// TwinCAT 3 PLC project Tc_Math
// Title: Tc_Math
// Company: NewEngineer
// Author: https://github.com/phucpha
// ProjectVersion: 1.1.2.0
// Description: this is library expand the Tc2_math
// ProgramVersion: 3.1.4024.0
// libraries:
//   Tc2_Math, * (Beckhoff Automation GmbH)
//   Tc2_Standard, * (Beckhoff Automation GmbH)
//   Tc2_System, * (Beckhoff Automation GmbH)
//   Tc2_Utilities, * (Beckhoff Automation GmbH)
//   Tc3_Module, * (Beckhoff Automation GmbH)
// project tree:
//   DUTs/ E_CompareTime.TcDUT
//   FCs/ F_CompareTime.TcPOU, FUN_Ceil.TcPOU, F_CheckInRange.TcPOU (not stored), F_CubicFit.TcPOU, F_CubitCalculate.TcPOU (not stored), F_InRange.TcPOU (not stored), F_QuanDraticCalculate.TcPOU (not stored), F_QuandraticFomularMaxValue.TcPOU, F_RoundLrealEx.TcPOU, F_ScaleValue.TcPOU (not stored)
//   / PlcTask.TcTTO
//   POUs/ FB_CalCulateAccumulation.TcPOU, FB_Derivative.TcPOU (not stored)
//   POUs/FIFO/ FB_FIFO_Lreal.TcPOU, FB_FIFO_TimeStruct.TcPOU, FB_Universal_FIFO.TcPOU, I_FIFO_Lreal.TcIO, I_FIFO_Timestruct.TcIO, I_Universal_FIFO.TcIO
// real-time tasks:
//   TASK PlcTask: cycle T#10ms, priority 20, ADS port 350

CONFIGURATION Tc_Math
    RESOURCE PLC ON TwinCAT3
        TASK PlcTask(INTERVAL := T#10ms, PRIORITY := 20);
    END_RESOURCE
END_CONFIGURATION

// ---- DUTs/E_CompareTime.TcDUT
{attribute 'strict'}
TYPE E_CompareTime :
(
	INVALID_PRE_TIME := 0,
	NEW_MINUTE := 5,
	NEW_HOUR := 10,
	NEW_DAY	:= 20,
	NEW_MONTH := 30,
	NEW_YEAR	:= 32,
	SAME_MINUTE := 35,
	SAME_HOUR := 40,
	SAME_DAY := 50,
	SAME_MONTH := 60,
	SAME_YEAR  := 70
);
END_TYPE

// ---- POUs/FIFO/I_FIFO_Lreal.TcIO
INTERFACE I_FIFO_Lreal EXTENDS I_Universal_FIFO

METHOD MR_AddValue : BOOL
VAR_INPUT
		Value : LREAL;
END_VAR
END_METHOD

PROPERTY oOldestValue : Lreal
GET
END_GET
END_PROPERTY

END_INTERFACE

// ---- POUs/FIFO/I_FIFO_Timestruct.TcIO
INTERFACE I_FIFO_Timestruct EXTENDS I_Universal_FIFO

METHOD MR_AddValue : BOOL
VAR_INPUT
		Value : TIMESTRUCT;
END_VAR
END_METHOD

PROPERTY oOldestValue : TIMESTRUCT
GET
END_GET
END_PROPERTY

END_INTERFACE

// ---- POUs/FIFO/I_Universal_FIFO.TcIO
INTERFACE I_Universal_FIFO

PROPERTY DataReady : bool
GET
END_GET
END_PROPERTY

PROPERTY HeadIndex : Uint
GET
END_GET
END_PROPERTY

PROPERTY IsEmpty : bool
GET
END_GET
END_PROPERTY

PROPERTY IsFull : bool
GET
END_GET
END_PROPERTY

METHOD MR_AckGetValue : BOOL
VAR_INPUT
END_VAR
END_METHOD

METHOD MR_Reset : BOOL
VAR_INPUT
END_VAR
END_METHOD

PROPERTY TailIndex : Uint
GET
END_GET
END_PROPERTY

END_INTERFACE

// ---- FCs/F_CompareTime.TcPOU
FUNCTION F_CompareTime : E_CompareTime
VAR_INPUT
		timestruct1 : TIMESTRUCT;//TIMEPREVIOUS
		timestruct2 : TIMESTRUCT;// TIME NOW
END_VAR
VAR_OUTPUT
	eCpMinute	: E_CompareTime;
	eCpHour		: E_CompareTime;
	eCpDay		: E_CompareTime;
	eCpMonth	: E_CompareTime;
	ecpYear		: E_CompareTime;
END_VAR

IF timestruct1.wYear < timestruct2.wYear THEN
	F_CompareTime := NEW_YEAR;
	ecpYear := NEW_YEAR;
	eCpMonth := NEW_MONTH;
	eCpDay := NEW_DAY;
	eCpHour := NEW_HOUR;
	eCpMinute := NEW_MINUTE;
ELSIF timestruct1.wYear > timestruct2.wYear THEN
		F_CompareTime := INVALID_PRE_TIME;
ELSE 
	ecpYear := SAME_YEAR;
	IF timestruct1.wMonth < timestruct2.wMonth THEN
		F_CompareTime := NEW_MONTH;
		eCpMonth := NEW_MONTH;
		eCpDay := NEW_DAY;
		eCpHour := NEW_HOUR;
		eCpMinute := NEW_MINUTE;
	ELSIF  timestruct1.wMonth > timestruct2.wMonth THEN
			F_CompareTime := INVALID_PRE_TIME;
	ELSE
		eCpMonth := SAME_MONTH;
		IF timestruct1.wDay < timestruct2.wDay THEN
			F_CompareTime := NEW_DAY;
			eCpDay := NEW_DAY;
			eCpHour := NEW_HOUR;
			eCpMinute := NEW_MINUTE;
		ELSIF timestruct1.wDay > timestruct2.wDay THEN
			F_CompareTime := INVALID_PRE_TIME;
		ELSE 
			eCpDay := SAME_DAY;
			IF timestruct1.wHour < timestruct2.wHour THEN
				F_CompareTime := NEW_HOUR;
				eCpHour := NEW_HOUR;
				eCpMinute := NEW_MINUTE;
			ELSIF timestruct1.wHour > timestruct2.wHour THEN
				F_CompareTime := INVALID_PRE_TIME; 
			ELSE
				eCpHour := SAME_HOUR;
				IF timestruct1.wMinute < timestruct2.wMinute THEN
					F_CompareTime := NEW_MINUTE;
					eCpMinute := NEW_MINUTE;
				ELSIF timestruct1.wMinute > timestruct2.wMinute THEN
					F_CompareTime := INVALID_PRE_TIME; 
				ELSE
					F_CompareTime := SAME_MINUTE;	
					eCpMinute := SAME_MINUTE;
			END_IF
			END_IF
		END_IF

	END_IF
END_IF

END_FUNCTION

// ---- FCs/FUN_Ceil.TcPOU
(* 
:Description: This function determines a integral value from a floating point number that is a fraction bigger than or equal that number
*)
FUNCTION FUN_Ceil : LREAL
VAR_INPUT
	lrValue : LREAL; (* Input value to round*)
END_VAR
VAR
	lrIntegral	: LREAL; (* Integral part of input value *)
	lrDecimal 	: LREAL; (* Decimal part of input value *)
END_VAR

(* Get integral part *)
lrIntegral := TRUNC(lrValue);

(* Get decimal part *)
lrDecimal := FRAC(lrValue);

(*Check decimal value and set final result *)
IF lrDecimal <> 0.0 THEN
	FUN_Ceil := lrIntegral + 1.0;
ELSE
	FUN_Ceil := lrIntegral;
END_IF

END_FUNCTION

// ---- FCs/F_CubicFit.TcPOU
FUNCTION F_CubicFit : BOOL
VAR_INPUT
    x : ARRAY[0..3] OF REAL; // x0, x1, x2, x3
    y : ARRAY[0..3] OF REAL; // y0, y1, y2, y3
END_VAR

VAR_OUTPUT
    a, b, c, d : REAL; // Polynomial coefficients
END_VAR

VAR
    Arr : ARRAY[0..3] OF ARRAY [0..4] OF REAL; // Augmented matrix (4x5)
    i, j, k : INT;
    factor : REAL;
END_VAR

// Build the augmented matrix A
FOR i := 0 TO 3 DO
    Arr[i][0] := x[i] * x[i] * x[i]; // x^3
    Arr[i][1] := x[i] * x[i];        // x^2
    Arr[i][2] := x[i];               // x
    Arr[i][3] := 1.0;                // constArrnt
    Arr[i][4] := y[i];               // y value (RHS)
END_FOR

// Gauss-Jordan Elimination
FOR i := 0 TO 3 DO
    // Normalize row i
    factor := Arr[i][ i];
    FOR j := i TO 4 DO
		IF NOT (-0.00000001 < factor  AND factor <  0.00000001) THEN
        	Arr[i][j] := Arr[i][ j] / factor;
		END_IF
    END_FOR

    // Eliminate other rows
    FOR k := 0 TO 3 DO
        IF k <> i THEN
            factor := Arr[k][ i];
            FOR j := i TO 4 DO
                Arr[k][j] := Arr[k][ j] - factor * Arr[i][j];
            END_FOR
        END_IF
    END_FOR
END_FOR

// Extract coefficients
a := Arr[0][ 4];
b := Arr[1][ 4];
c := Arr[2][ 4];
d := Arr[3][ 4];

END_FUNCTION

// ---- FCs/F_QuandraticFomularMaxValue.TcPOU
FUNCTION F_QuandraticFomularMaxValue : LREAL 
VAR_INPUT
	A : LREAL;
	B : LREAL;
	C : LREAL;
	xLimit1 : LREAL;
	xLimit2 : LREAL;
END_VAR
VAR
	yAtxLimit1 : LREAL;
	yAtxLimit2 : LREAL;
	Adot : LREAL; // Adot = A'
	Bdot : LREAL; // Bdot = B'
	x : LREAL;
END_VAR
VAR_OUTPUT
	MaxValue : LREAL;
END_VAR

yAtxLimit1 := F_QuanDraticCalculate(
	A := A,
	B := B,
	C := C,
	x := xLimit1
);
yAtxLimit2 := F_QuanDraticCalculate(
	A := A,
	B := B,
	C := C,
	x := xLimit2
);		
IF A > 0 THEN
	MaxValue := MAX(yAtxLimit1, yAtxLimit2);
ELSIF A < 0 THEN
	Adot := 2 * A;
	Bdot := B;
	x := -Bdot / Adot;
	MaxValue := F_QuanDraticCalculate(
		A := A,
		B := B,
		C := C,
		x := x
	);	
ELSE // A = 0, b is any
	MaxValue := MAX(yAtxLimit1, yAtxLimit2);
END_IF
F_QuandraticFomularMaxValue := MaxValue;

END_FUNCTION

// ---- FCs/F_RoundLrealEx.TcPOU
FUNCTION F_RoundLrealEx : LREAL
VAR_INPUT
	lrIn : LREAL;
	iPrecision : UINT;
END_VAR
VAR
	lrTemp	: LREAL;
END_VAR

lrTemp := lrIn * EXPT(10,iPrecision);
lrTemp := LTRUNC(lrTemp);
F_RoundLrealEx := lrTemp / EXPT(10,iPrecision);

END_FUNCTION

// ---- POUs/FB_CalCulateAccumulation.TcPOU
(* Will be refactor later
| need refactor to independence to fbMachineTime 
*)
FUNCTION_BLOCK FB_CalCulateAccumulation
VAR_INPUT
	lrAccumulator : LREAL  := 0;
	CurrentTime : TIMESTRUCT; 
END_VAR
VAR_OUTPUT
	accumulatedValueOut : LREAL;// value = lrAccumulator(timeNew) - lrAccumulator(timeOld)
	previousTimestampOut : TIMESTRUCT;// TimeOld
	bNewPeriodAlarm : BOOL;// Remain True in 30s if not be ackNowledge
	
END_VAR
VAR

	
	eCpHour		: E_CompareTime;
	eCpDay 		: E_CompareTime;
	eCpMonth	: E_CompareTime;
	eCpYear		: E_CompareTime;
	eCpMinute	: E_CompareTime;
	eSameTime : E_CompareTime;
	eNewTime : E_CompareTime;
	eRfTimeCompare : REFERENCE TO E_CompareTime;
	sName 		: STRING;
	eState : UINT;
	TonRemainOutput : TON;
	eTimeAccumulate : E_CompareTime;
	bInit : BOOL;
	bReset : BOOL;
	bRequestUpdate_ValueInLastTime: BOOL;
END_VAR

VAR PERSISTENT 
	bUpdatedValueLastHour : BOOL;// reject Power OFF unexpected
	previousTimestamp	: TIMESTRUCT;
	ValueInLastTime : LREAL;
	accumulatedValue : LREAL;
	
	
END_VAR
VAR CONSTANT
	eStateUinitialized : UINT := 0;
	eStateInit : UINT := 10;
	eStateRun : UINT := 20;
	eStateReset : UINT := 100;
	TimeNewPeriodAlarm : TIME := T#30s;
END_VAR

CASE eState OF
	eStateUinitialized: // unInitialized
		;// will go to eStateInit if MR_Run is called 
		
	eStateInit: 
		;// will call by MR_Init
		
	eStateRun: //StateRun
		MS_Run();
		
	eStateReset :
		MS_Reset();
END_CASE

IF eState > 0 AND bReset THEN
	eState := eStateReset;
END_IF

PROPERTY isInitDone : bool
GET
END_GET
END_PROPERTY

PROPERTY isRuning : bool
GET
isRuning := eState = eStateRun;
END_GET
END_PROPERTY

// if not return true , check the Current time and PreviousTime in fb
METHOD MR_Acknowledge : BOOL
VAR_INPUT
END_VAR
bNewPeriodAlarm := FALSE;
IF eRfTimeCompare = eSameTime THEN
	MR_Acknowledge := TRUE;
END_IF
END_METHOD

METHOD MR_Init : BOOL
VAR_INPUT
END_VAR
IF eState = eStateUinitialized THEN// init;
	bInit := true;
	IF MS_Init() THEN
		MR_Init := TRUE;
		eState := eStateRun;
	END_IF
END_IF
END_METHOD

METHOD MR_Reset : BOOL
VAR_INPUT
END_VAR
bReset := TRUE;
IF eState = eStateUinitialized THEN
	MR_Reset := TRUE;
	bReset := false;
END_IF
END_METHOD

METHOD Protected MS_Init : BOOL
VAR_INPUT
END_VAR
CASE eTimeAccumulate OF
	NEW_MINUTE :
		eSameTime := SAME_MINUTE;
		eNewTime := NEW_MINUTE;
		eRfTimeCompare REF= eCpMinute;
		MS_Init := TRUE;
	NEW_HOUR :
		eSameTime := SAME_HOUR;
		eNewTime := NEW_HOUR;
		eRfTimeCompare REF= eCpHour;
		MS_Init := TRUE;
	NEW_DAY	:
		eSameTime := SAME_DAY;
		eNewTime := NEW_DAY;
		eRfTimeCompare REF= eCpDay;
		MS_Init := TRUE;
	NEW_MONTH:
		eSameTime := SAME_MONTH;
		eNewTime := NEW_MONTH;
		eRfTimeCompare REF= eCpMonth;
		MS_Init := TRUE;
	NEW_YEAR:
		eSameTime := SAME_YEAR;
		eNewTime := NEW_YEAR;
		eRfTimeCompare REF= eCpYear;
		MS_Init := true;
END_CASE
END_METHOD

METHOD protected MS_Reset : BOOL
VAR_INPUT
END_VAR
//retainvalue
	
	bUpdatedValueLastHour := FALSE;
	previousTimestamp.wYear := 0;
	previousTimestamp.wMonth := 0;
	previousTimestamp.wDay := 0;
	previousTimestamp.wMinute := 0;
	previousTimestamp.wSecond := 0;
	previousTimestamp.wMilliseconds := 0;
	ValueInLastTime := 0 ;
	accumulatedValue := 0 ;
// out_put
	accumulatedValueOut := 0;
	previousTimestampOut.wYear := 0;
	previousTimestampOut.wMonth := 0;
	previousTimestampOut.wDay := 0;
	previousTimestampOut.wMinute := 0;
	previousTimestampOut.wSecond := 0;
	previousTimestampOut.wMilliseconds := 0;
	bNewPeriodAlarm := false;// Remain True 
	
// 	RETURN TO uninit
	eState := eStateUinitialized;
	eRfTimeCompare REF= 0;
END_METHOD

METHOD Protected MS_Run : BOOL
VAR_INPUT
END_VAR
F_CompareTime( 
	timestruct1 := previousTimestamp,
	timestruct2 := CurrentTime,
	eCpMinute => eCpMinute, 
	eCpHour => eCpHour,
	eCpDay => eCpDay,
	eCpMonth => eCpMonth,
	ecpYear => eCpYear
);

IF eRfTimeCompare = eNewTime THEN
	// update to output
	accumulatedValueOut := accumulatedValue;
	previousTimestampOut := previousTimestamp;
	bNewPeriodAlarm := TRUE;
	// update the the last hour and time
	bUpdatedValueLastHour := FALSE;
	IF lrAccumulator > 0.1 THEN
		ValueInLastTime := lrAccumulator;
		bRequestUpdate_ValueInLastTime := FALSE;
		// UpdateOK
		bUpdatedValueLastHour := TRUE;
	ELSE
		bRequestUpdate_ValueInLastTime := TRUE;
	END_IF
	ValueInLastTime := lrAccumulator;
	previousTimestamp := CurrentTime;


ELSIF eRfTimeCompare = eSameTime AND bUpdatedValueLastHour THEN
	IF lrAccumulator > 0.1 THEN // reject the situation that just TURN ON IPC so lrAccumulator = -8888888888888888.444444444444
		accumulatedValue := lrAccumulator - ValueInLastTime;
	END_IF
ELSIF eRfTimeCompare = eSameTime AND NOT bUpdatedValueLastHour THEN
	ValueInLastTime := lrAccumulator;
	previousTimestamp := CurrentTime;
ELSE
	; //invalid time Compare


END_IF
	
TonRemainOutput( IN := bNewPeriodAlarm , PT := TimeNewPeriodAlarm);

IF TonRemainOutput.Q THEN
	bNewPeriodAlarm := false;
END_IF
IF bRequestUpdate_ValueInLastTime THEN
	IF lrAccumulator > 0.1 THEN
		ValueInLastTime := lrAccumulator;
		bRequestUpdate_ValueInLastTime := FALSE;
		// UpdateOK
		bUpdatedValueLastHour := TRUE;
	END_IF
END_IF
END_METHOD

PROPERTY Name : string
GET
Name := sName;
END_GET
SET
sName := Name;
END_SET
END_PROPERTY

// Set TimeAccumulate before call Mr_Init.
//NEW_MINUTE := 5,
//	NEW_HOUR := 10,
//	NEW_DAY	:= 20,
//	NEW_MONTH := 30,
//	NEW_YEAR	:= 32,
PROPERTY TimeAccumulate : E_CompareTime
GET
TimeAccumulate := eTimeAccumulate;
END_GET
SET
eTimeAccumulate := TimeAccumulate;
END_SET
END_PROPERTY

END_FUNCTION_BLOCK

// ---- POUs/FIFO/FB_FIFO_Lreal.TcPOU
FUNCTION_BLOCK FB_FIFO_Lreal EXTENDS FB_Universal_FIFO IMPLEMENTS I_FIFO_Lreal
VAR_OUTPUT
	OldestData : LREAL;
END_VAR
VAR PERSISTENT
	Queue : ARRAY[0..MaxQueueSize-1] OF LREAL;  // FIFO queue (size is 100 elements)
END_VAR



//    // Log new data only if LogData is TRUE
//    IF rTrigLogData.Q THEN
//        IF Count < MaxQueueSize THEN
//            Queue[Head] := NewEnergyData;
//            Head := (Head + 1) MOD MaxQueueSize;
//            Count := Count + 1;
//        ELSE
//            // FIFO is full, overwrite old data if needed
//            Tail := (Tail + 1) MOD MaxQueueSize;
//            Queue[Head] := NewEnergyData;
//            Head := (Head + 1) MOD MaxQueueSize;
//            // Tail position is updated
//        END_IF
//        DataReady := TRUE;  // New data is now ready to be processed
     
//    END_IF

    // Retrieve and manage oldest data for processing

// if dataready return true, else return false
METHOD  MR_AckGetValue : BOOL
VAR_INPUT
END_VAR
SUPER^.MR_AckGetValue();
  OldestData := Queue[Tail];
 MR_AckGetValue := true;
END_METHOD

METHOD MR_AddValue : BOOL
VAR_INPUT
		Value : LREAL;
END_VAR
  IF Count < MaxQueueSize THEN
            Queue[Head] := Value;
            Head := (Head + 1) MOD MaxQueueSize;
            Count := Count + 1;
  ELSE
            // FIFO is full, overwrite old data if needed
            Tail := (Tail + 1) MOD MaxQueueSize;
            Queue[Head] := Value;
            Head := (Head + 1) MOD MaxQueueSize;
            // Tail position is updated
			
  END_IF
  
  OldestData := Queue[Tail];
  bDataReady := TRUE; 
  
  
  MR_AddValue := true;
END_METHOD

// need overide to reset oldestValue
METHOD MR_Reset : BOOL
VAR_INPUT
END_VAR
SUPER^.MR_Reset();
OldestData := 0;
MR_Reset := true;
END_METHOD

PROPERTY oOldestValue : Lreal
GET
oOldestValue := OldestData;
END_GET
END_PROPERTY

END_FUNCTION_BLOCK

// ---- POUs/FIFO/FB_Universal_FIFO.TcPOU
FUNCTION_BLOCK ABSTRACT FB_Universal_FIFO IMPLEMENTS I_Universal_FIFO

VAR PERSISTENT    
	//Queue : ARRAY[0..MaxQueueSize-1] OF REAL;  // FIFO queue (size is 100 elements)
    Head : UINT := 0;  // Points to the next position to store data
    Tail : UINT := 0;  // Points to the oldest data position
    Count : UINT := 0;  // Number of elements currently in the FIFO
	bDataReady : BOOL; 
	eState : UINT;
END_VAR

VAR CONSTANT
	MaxQueueSize : UINT := 255;  // Number of elements in the FIFO queue

END_VAR

VAR_OUTPUT

   
END_VAR

PROPERTY CurrentCount : Uint
GET
CurrentCount := Count;
END_GET
END_PROPERTY

PROPERTY DataReady : BOOL
GET
DataReady := bDataReady;
END_GET
END_PROPERTY

PROPERTY HeadIndex : UINT
GET
HeadIndex := Head;
END_GET
END_PROPERTY

PROPERTY IsEmpty : bool
GET
IF Count = 0 THEN
	IsEmpty := TRUE;
ELSE
	IsEmpty := false;
END_IF
END_GET
END_PROPERTY

PROPERTY IsFull : bool
GET
IF count = MaxQueueSize THEN
	IsFull := TRUE;
ELSE 
	IsFull := FALSE;
END_IF
END_GET
END_PROPERTY

// if dataready return true, else return false// need overiding a part
METHOD MR_AckGetValue : BOOL
VAR_INPUT
END_VAR
IF bDataReady THEN
      
            // Data has been processed, so move to the next item in the queue
            Tail := (Tail + 1) MOD MaxQueueSize;
            Count := Count - 1;
            IF Count = 0 THEN
                bDataReady := FALSE;  // No more data to process
            END_IF
        
            // Data is still ready to be processed
        
    MR_AckGetValue := TRUE;   
ELSE 
	MR_AckGetValue := FALSE;
END_IF
// set oldest value in child fb here
// OldestData :=   Queue[Tail];
/////
END_METHOD

// need overide to reset oldestValue
METHOD MR_Reset : BOOL
VAR_INPUT
END_VAR
     Head := 0;
     Tail := 0;
     Count := 0;
	 bDataReady := FALSE;
	 MR_Reset := TRUE;
END_METHOD

PROPERTY TailIndex : Uint
GET
TailIndex := Tail;
END_GET
END_PROPERTY

END_FUNCTION_BLOCK

// ---- POUs/FIFO/FB_FIFO_TimeStruct.TcPOU
FUNCTION_BLOCK FB_FIFO_TimeStruct EXTENDS FB_Universal_FIFO IMPLEMENTS I_FIFO_Timestruct
VAR_INPUT
END_VAR
VAR_OUTPUT
END_VAR
VAR_OUTPUT
	OldestData : TIMESTRUCT;
END_VAR
VAR PERSISTENT
	Queue : ARRAY[0..MaxQueueSize-1] OF TIMESTRUCT;  // FIFO queue (size is 100 elements)
END_VAR
VAR CONSTANT
	timstructZero : TIMESTRUCT;
END_VAR

// if dataready return true, else return false
METHOD  MR_AckGetValue : BOOL
VAR_INPUT
END_VAR
SUPER^.MR_AckGetValue();
  OldestData := Queue[Tail];
 MR_AckGetValue := true;
END_METHOD

METHOD MR_AddValue : BOOL
VAR_INPUT
		Value : TIMESTRUCT;
END_VAR
  IF Count < MaxQueueSize THEN
            Queue[Head] := Value;
            Head := (Head + 1) MOD MaxQueueSize;
            Count := Count + 1;
  ELSE
            // FIFO is full, overwrite old data if needed
            Tail := (Tail + 1) MOD MaxQueueSize;
            Queue[Head] := Value;
            Head := (Head + 1) MOD MaxQueueSize;
            // Tail position is updated
			
  END_IF
  
  OldestData := Queue[Tail];
  bDataReady := TRUE; 
  
  
  MR_AddValue := true;
END_METHOD

// need overide to reset oldestValue
METHOD MR_Reset : BOOL
VAR_INPUT
END_VAR
SUPER^.MR_Reset();
OldestData := timstructZero;
MR_Reset := true;
END_METHOD

PROPERTY oOldestValue : TIMESTRUCT
GET
oOldestValue := OldestData;
END_GET
END_PROPERTY

END_FUNCTION_BLOCK
